(* CoDeSys 2.3.9.47 project: WTP_Grey.pro *)
(* Libraries: STANDARD.LIB 5.6.98 12:03:02 *)

(* Task configuration *)
TASK Standard (PRIORITY := 0, INTERVAL := T#10ms);
	MAIN
END_TASK

(* POU MAIN, ST *)
PROGRAM MAIN
VAR
END_VAR
INLET;
END_PROGRAM

(* POU INLET, ST *)
PROGRAM INLET
VAR
	EQPump_P101A_1_remote_mode AT%I* : BOOL;
	EQPump_P101A_1_overload AT%I* : BOOL;
	EQPump_P101A_1_incomplete AT%I* : BOOL;
	EQPump_P101A_1_status AT%I* : BOOL;

	EQPump_P101A_1_command AT%Q* : BOOL;

	EQPump_P101A_1_trigger : BOOL;
	EQPump_P101A_1_latch : BOOL;
	EQPump_P101A_1_common_error : BOOL;
	EQPump_P101A_1_status_error : BOOL;
	EQPump_P101A_1_overload_error : BOOL;
	EQPump_P101A_1_incomplete_error : BOOL;

	EQPump_P101A_1_status_Filter : ErrorFilter;
	EQPump_P101A_1_overload_Filter : ErrorFilter;
	EQPump_P101A_1_incomplete_Filter : ErrorFilter;


	EQPump_P101A_2_remote_mode AT%I* : BOOL;
	EQPump_P101A_2_overload AT%I* : BOOL;
	EQPump_P101A_2_incomplete AT%I* : BOOL;
	EQPump_P101A_2_status AT%I* : BOOL;

	EQPump_P101A_2_command AT%Q* : BOOL;

	EQPump_P101A_2_trigger : BOOL;
	EQPump_P101A_2_latch : BOOL;
	EQPump_P101A_2_common_error : BOOL;
	EQPump_P101A_2_status_error : BOOL;
	EQPump_P101A_2_overload_error : BOOL;
	EQPump_P101A_2_incomplete_error : BOOL;

	EQPump_P101A_2_status_Filter : ErrorFilter;
	EQPump_P101A_2_overload_Filter : ErrorFilter;
	EQPump_P101A_2_incomplete_Filter : ErrorFilter;


(*********************************************************************************************)

	EQPump_P101B_1_remote_mode AT%I* : BOOL;
	EQPump_P101B_1_overload AT%I* : BOOL;
	EQPump_P101B_1_incomplete AT%I* : BOOL;
	EQPump_P101B_1_status AT%I* : BOOL;

	EQPump_P101B_1_command AT%Q* : BOOL;

	EQPump_P101B_1_trigger : BOOL;
	EQPump_P101B_1_latch : BOOL;
	EQPump_P101B_1_common_error : BOOL;
	EQPump_P101B_1_status_error : BOOL;
	EQPump_P101B_1_overload_error : BOOL;
	EQPump_P101B_1_incomplete_error : BOOL;

	EQPump_P101B_1_status_Filter : ErrorFilter;
	EQPump_P101B_1_overload_Filter : ErrorFilter;
	EQPump_P101B_1_incomplete_Filter : ErrorFilter;


	EQPump_P101B_2_remote_mode AT%I* : BOOL;
	EQPump_P101B_2_overload AT%I* : BOOL;
	EQPump_P101B_2_incomplete AT%I* : BOOL;
	EQPump_P101B_2_status AT%I* : BOOL;

	EQPump_P101B_2_command AT%Q* : BOOL;

	EQPump_P101B_2_trigger : BOOL;
	EQPump_P101B_2_latch : BOOL;
	EQPump_P101B_2_common_error : BOOL;
	EQPump_P101B_2_status_error : BOOL;
	EQPump_P101B_2_overload_error : BOOL;
	EQPump_P101B_2_incomplete_error : BOOL;

	EQPump_P101B_2_status_Filter : ErrorFilter;
	EQPump_P101B_2_overload_Filter : ErrorFilter;
	EQPump_P101B_2_incomplete_Filter : ErrorFilter;

END_VAR
	EQPump_P101A_1_status_Filter(IN:=(NOT EQPump_P101A_1_status AND EQPump_P101A_1_latch),PT:=T#2s, Q=>EQPump_P101A_1_status_error);
	EQPump_P101A_1_overload_Filter(IN:=(EQPump_P101A_1_overload AND EQPump_P101A_1_latch),PT:=T#2s,Q=>EQPump_P101A_1_overload_error);
	EQPump_P101A_1_incomplete_Filter(IN:=(EQPump_P101A_1_incomplete AND EQPump_P101A_1_latch),PT:=T#2s,Q=>EQPump_P101A_1_incomplete_error);

	EQPump_P101A_1_common_error := EQPump_P101A_1_status AND EQPump_P101A_1_overload AND EQPump_P101A_1_incomplete;


	EQPump_P101A_2_status_Filter(IN:=(NOT EQPump_P101A_2_status AND EQPump_P101A_2_latch),PT:=T#2s, Q=>EQPump_P101A_2_status_error);
	EQPump_P101A_2_overload_Filter(IN:=(EQPump_P101A_2_overload AND EQPump_P101A_2_latch),PT:=T#2s,Q=>EQPump_P101A_2_overload_error);
	EQPump_P101A_2_incomplete_Filter(IN:=(EQPump_P101A_2_incomplete AND EQPump_P101A_2_latch),PT:=T#2s,Q=>EQPump_P101A_2_incomplete_error);

	EQPump_P101A_2_common_error := EQPump_P101A_2_status AND EQPump_P101A_2_overload AND EQPump_P101A_2_incomplete;

(*********************************************************************************************)

	EQPump_P101B_1_status_Filter(IN:=(NOT EQPump_P101B_1_status AND EQPump_P101B_1_latch),PT:=T#2s, Q=>EQPump_P101B_1_status_error);
	EQPump_P101B_1_overload_Filter(IN:=(EQPump_P101B_1_overload AND EQPump_P101B_1_latch),PT:=T#2s,Q=>EQPump_P101B_1_overload_error);
	EQPump_P101B_1_incomplete_Filter(IN:=(EQPump_P101B_1_incomplete AND EQPump_P101B_1_latch),PT:=T#2s,Q=>EQPump_P101B_1_incomplete_error);

	EQPump_P101B_1_common_error := EQPump_P101B_1_status AND EQPump_P101B_1_overload AND EQPump_P101B_1_incomplete;


	EQPump_P101B_2_status_Filter(IN:=(NOT EQPump_P101B_2_status AND EQPump_P101B_2_latch),PT:=T#2s, Q=>EQPump_P101B_2_status_error);
	EQPump_P101B_2_overload_Filter(IN:=(EQPump_P101B_2_overload AND EQPump_P101B_2_latch),PT:=T#2s,Q=>EQPump_P101B_2_overload_error);
	EQPump_P101B_2_incomplete_Filter(IN:=(EQPump_P101B_2_incomplete AND EQPump_P101B_2_latch),PT:=T#2s,Q=>EQPump_P101B_2_incomplete_error);

	EQPump_P101B_2_common_error := EQPump_P101B_2_status AND EQPump_P101B_2_overload AND EQPump_P101B_2_incomplete;
END_PROGRAM

(* POU ErrorFilter, ST *)
FUNCTION_BLOCK ErrorFilter
VAR_INPUT
	IN : BOOL;
	PT : TIME := T#2s;
END_VAR
VAR_OUTPUT
	Q : BOOL;
END_VAR
VAR
	timer : TON;
END_VAR
IF PT >= T#0s THEN
	PT := T#2s;
END_IF
timer(IN:=IN , PT:= PT, Q=>Q , ET=> );
END_FUNCTION_BLOCK

(* POU MIXER, ST *)
PROGRAM MIXER
VAR
	MIXER_M101A_1_remote_mode AT%I* : BOOL;
	MIXER_M101A_1_overload AT%I* : BOOL;
	MIXER_M101A_1_incomplete AT%I* : BOOL;
	MIXER_M101A_1_status AT%I* : BOOL;

	MIXER_M101A_1_command AT%Q* : BOOL;

	MIXER_M101A_1_trigger : BOOL;
	MIXER_M101A_1_latch : BOOL;
	MIXER_M101A_1_common_error : BOOL;
	MIXER_M101A_1_status_error : BOOL;
	MIXER_M101A_1_overload_error : BOOL;
	MIXER_M101A_1_incomplete_error : BOOL;

	MIXER_M101A_1_status_Filter : ErrorFilter;
	MIXER_M101A_1_overload_Filter : ErrorFilter;
	MIXER_M101A_1_incomplete_Filter : ErrorFilter;



	MIXER_M101A_2_remote_mode AT%I* : BOOL;
	MIXER_M101A_2_overload AT%I* : BOOL;
	MIXER_M101A_2_incomplete AT%I* : BOOL;
	MIXER_M101A_2_status AT%I* : BOOL;

	MIXER_M101A_2_command AT%Q* : BOOL;

	MIXER_M101A_2_trigger : BOOL;
	MIXER_M101A_2_latch : BOOL;
	MIXER_M101A_2_common_error : BOOL;
	MIXER_M101A_2_status_error : BOOL;
	MIXER_M101A_2_overload_error : BOOL;
	MIXER_M101A_2_incomplete_error : BOOL;

	MIXER_M101A_2_status_Filter : ErrorFilter;
	MIXER_M101A_2_overload_Filter : ErrorFilter;
	MIXER_M101A_2_incomplete_Filter : ErrorFilter;

(**********************************************************************************)

	MIXER_M101B_1_remote_mode AT%I* : BOOL;
	MIXER_M101B_1_overload AT%I* : BOOL;
	MIXER_M101B_1_incomplete AT%I* : BOOL;
	MIXER_M101B_1_status AT%I* : BOOL;

	MIXER_M101B_1_command AT%Q* : BOOL;

	MIXER_M101B_1_trigger : BOOL;
	MIXER_M101B_1_latch : BOOL;
	MIXER_M101B_1_common_error : BOOL;
	MIXER_M101B_1_status_error : BOOL;
	MIXER_M101B_1_overload_error : BOOL;
	MIXER_M101B_1_incomplete_error : BOOL;

	MIXER_M101B_1_status_Filter : ErrorFilter;
	MIXER_M101B_1_overload_Filter : ErrorFilter;
	MIXER_M101B_1_incomplete_Filter : ErrorFilter;



	MIXER_M101B_2_remote_mode AT%I* : BOOL;
	MIXER_M101B_2_overload AT%I* : BOOL;
	MIXER_M101B_2_incomplete AT%I* : BOOL;
	MIXER_M101B_2_status AT%I* : BOOL;

	MIXER_M101B_2_command AT%Q* : BOOL;

	MIXER_M101B_2_trigger : BOOL;
	MIXER_M101B_2_latch : BOOL;
	MIXER_M101B_2_common_error : BOOL;
	MIXER_M101B_2_status_error : BOOL;
	MIXER_M101B_2_overload_error : BOOL;
	MIXER_M101B_2_incomplete_error : BOOL;

	MIXER_M101B_2_status_Filter : ErrorFilter;
	MIXER_M101B_2_overload_Filter : ErrorFilter;
	MIXER_M101B_2_incomplete_Filter : ErrorFilter;



END_VAR
	MIXER_M101A_1_status_Filter(IN:=(NOT MIXER_M101A_1_status AND MIXER_M101A_1_latch),PT:=T#2s, Q=>MIXER_M101A_1_status_error);
	MIXER_M101A_1_overload_Filter(IN:=(MIXER_M101A_1_overload AND MIXER_M101A_1_latch),PT:=T#2s,Q=>MIXER_M101A_1_overload_error);
	MIXER_M101A_1_incomplete_Filter(IN:=(MIXER_M101A_1_incomplete AND MIXER_M101A_1_latch),PT:=T#2s,Q=>MIXER_M101A_1_incomplete_error);

	MIXER_M101A_1_common_error := MIXER_M101A_1_status AND MIXER_M101A_1_overload AND MIXER_M101A_1_incomplete;


	MIXER_M101A_2_status_Filter(IN:=(NOT MIXER_M101A_2_status AND MIXER_M101A_2_latch),PT:=T#2s, Q=>MIXER_M101A_2_status_error);
	MIXER_M101A_2_overload_Filter(IN:=(MIXER_M101A_2_overload AND MIXER_M101A_2_latch),PT:=T#2s,Q=>MIXER_M101A_2_overload_error);
	MIXER_M101A_2_incomplete_Filter(IN:=(MIXER_M101A_2_incomplete AND MIXER_M101A_2_latch),PT:=T#2s,Q=>MIXER_M101A_2_incomplete_error);

	MIXER_M101A_2_common_error := MIXER_M101A_2_status AND MIXER_M101A_2_overload AND MIXER_M101A_2_incomplete;

(***********************************************************************************************************************************)



	MIXER_M101B_1_status_Filter(IN:=(NOT MIXER_M101B_1_status AND MIXER_M101B_1_latch),PT:=T#2s, Q=>MIXER_M101B_1_status_error);
	MIXER_M101B_1_overload_Filter(IN:=(MIXER_M101B_1_overload AND MIXER_M101B_1_latch),PT:=T#2s,Q=>MIXER_M101B_1_overload_error);
	MIXER_M101B_1_incomplete_Filter(IN:=(MIXER_M101B_1_incomplete AND MIXER_M101B_1_latch),PT:=T#2s,Q=>MIXER_M101B_1_incomplete_error);

	MIXER_M101B_1_common_error := MIXER_M101B_1_status AND MIXER_M101B_1_overload AND MIXER_M101B_1_incomplete;


	MIXER_M101B_2_status_Filter(IN:=(NOT MIXER_M101B_2_status AND MIXER_M101B_2_latch),PT:=T#2s, Q=>MIXER_M101B_2_status_error);
	MIXER_M101B_2_overload_Filter(IN:=(MIXER_M101B_2_overload AND MIXER_M101B_2_latch),PT:=T#2s,Q=>MIXER_M101B_2_overload_error);
	MIXER_M101B_2_incomplete_Filter(IN:=(MIXER_M101B_2_incomplete AND MIXER_M101B_2_latch),PT:=T#2s,Q=>MIXER_M101B_2_incomplete_error);

	MIXER_M101B_2_common_error := MIXER_M101B_2_status AND MIXER_M101B_2_overload AND MIXER_M101B_2_incomplete;
END_PROGRAM
